// TIA Portal V20 export
TYPE "UDT_Interlock_Enfardadora"
   STRUCT
      "ENTREGA ULMA A ENF" : Struct
         AVTF_ULMA_ENF : Bool;
         DESC_ACT_ULMA_ENF : Bool;
         MAN_AV_SIMUL_ULMA_ENF : Bool;
         MAN_RET_SIMUL_ULMA_ENF : Bool;
         PTF_ENF_ULMA : Bool;
         FTF_ENF_ULMA : Bool;
         MAN_AV_SIMUL_ENF_ULMA : Bool;
         MAN_RET_SIMUL_ENF_ULMA : Bool;
         Bit_0_Tipo_Enfardado : Bool;
         Bit_1_Tipo_Enfardado : Bool;
         Peticion_Acceso : Bool;
         Peticion_Rearme : Bool;
         Peticion_Marcha : Bool;
         Puerta_abierta : Bool;
         Byte1_bit6 : Bool;
         EMERGENCIA_ULMA : Bool;
      END_STRUCT;
      "ENTREGA ENF A ULMA" : Struct
         AVTF_ENF_ULMA : Bool;
         DESC_ACT_ENF_ULMA : Bool;
         MAN_AV_SIMUL_ENF_ULMA : Bool;
         MAN_RET_SIMUL_ENF_ULMA : Bool;
         PTF_ULMA_ENF : Bool;
         FTF_ULMA_ENF : Bool;
         MAN_AV_SIMUL_ULMA_ENF : Bool;
         MAN_RET_SIMUL_ULMA_ENF : Bool;
         Error_Enfardadora : Bool;
         Marcha_Enfardadora : Bool;
         Presencia_carga_Enfardadora : Bool;
         Permiso_Acceso_Recinto : Bool;
         Byte3_bit4 : Bool;
         Byte3_bit5 : Bool;
         Byte3_bit6 : Bool;
         PARADA_EMERGENCIA : Bool;
      END_STRUCT;
   END_STRUCT;
END_TYPE
